# B&R Automation Studio project Bnr-Testing
Automation Studio 4.6.3.55 SP

## Configuration Config1

CPU X20CP1586, AutomationRuntime B4.63, Build 4.1.2, Vc V4.62.0

### Task classes (Cpu.sw)
```
Cyclic#4:
  Program <- Program.prg
Cyclic#7:
  RevInfo <- RevInfo.RevInfo.prg
Libraries: AsBrStr
```

## Logical view

### RevInfo.var
```iecst
VAR CONSTANT
	revision : STRING[80] := 'f5992fa';
	revisionDate : STRING[80] := '2022-05-19 14:30:05 +0800';
	revisionAuthor : STRING[80] := 'Brian Ng';
	branchName : STRING[80] := 'HMI';
	uncommittedChanges : STRING[80] := ' 35 files changed, 2681 insertions(+), 150 deletions(-)';
	buildDate  : STRING[80] := '2022-05-19 15:58:43 +0800';
	buildConfiguration : STRING[80] := 'Config1';
	builder : STRING[80] := 'Brian Ng';
END_VAR
```

- Visualisation Logical/mappView (not shown)

### Program Logical/Program (ANSIC)

#### Main.c - Init, cyclic, exit code
```c
#include <bur/plctypes.h>
#ifdef _DEFAULT_INCLUDES
#include <AsDefault.h>
//constants//
#ifdef _REPLACE_CONST
#define MyConstant 123U
#else
_GLOBAL_CONST unsigned char MyConstant;
#endif

void _INIT ProgramInit(void)
{
	dummy = 1;
}

void _CYCLIC ProgramCyclic(void)
{

}

void _EXIT ProgramExit(void)
{

}
```

Listed in the project but not available here: Logical/Global.typ, Logical/Global.var, Logical/Libraries, Logical/Program/Types.typ, Logical/Program/Variables.var
